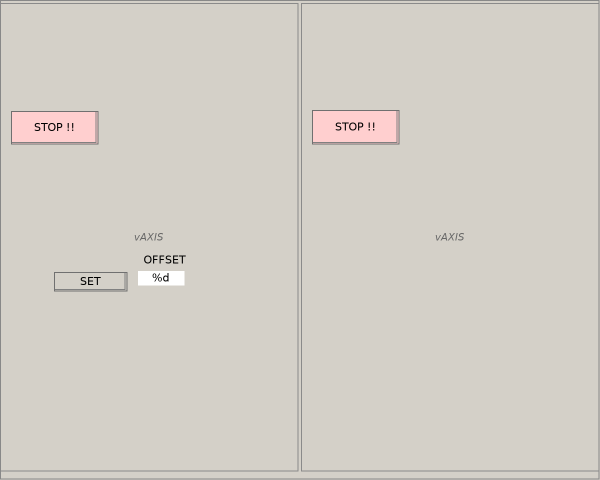
VISUALIZATION vAXES2  // 600x480
    Frame (0,3 298x468)
        shows vAXIS(vAxis := LIFT2)
    Frame (301,3 298x468)
        shows vAXIS(vAxis := XY2)
    Textfield (137,270 48x16), "%d", text variable: iOFFSET2
        OnMouseDown: write the text variable via Default
    Label (135,249 59x22), "OFFSET"
    Button (312,110 87x34), "STOP !!"
        OnMouseDown: execute { ACTION1.bSTOP_ALL:=TRUE; }
    Button (11,111 87x33), "STOP !!"
        OnMouseDown: execute { ACTION1.bSTOP_ALL:=TRUE; }
    Button (54,272 73x19), "SET"
        tap bWP_Start
END_VISUALIZATION

(* stored: Version 1.1.0.1, ProductVersion 3.1.4024.12
   Visu vAXES2: Id {8a8c1df9-6a38-4a54-a093-90621d7ed456} *)
